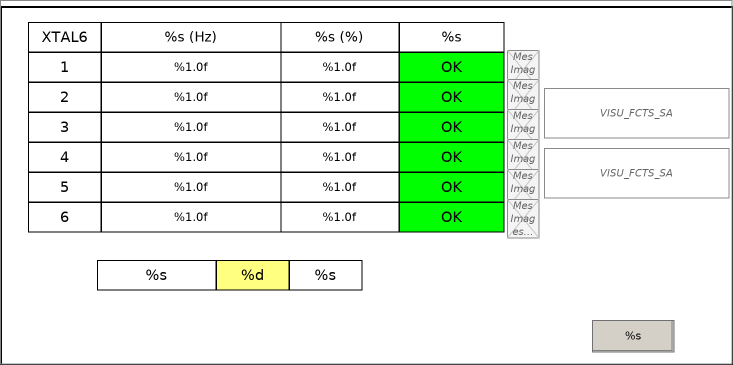
VISUALIZATION VISU_XTAL6_ZOOM  // 733x365, background image fond_blanc_1280_1024
VAR_IN_OUT
	m_Input_XTAL6 : BLOCK_XTAL6;
END_VAR
    Rectangle (0,6 733x359)
    RoundedRectangle (280,52 119x30), "%1.0f", text variable: m_Input_XTAL6.STATE_LIFE[1]
    RoundedRectangle (280,82 119x30), "%1.0f", text variable: m_Input_XTAL6.STATE_LIFE[2]
    RoundedRectangle (280,112 119x30), "%1.0f", text variable: m_Input_XTAL6.STATE_LIFE[3]
    RoundedRectangle (28,52 73x30), "1"
    RoundedRectangle (28,82 73x30), "2"
    RoundedRectangle (28,112 73x30), "3"
    RoundedRectangle (280,22 119x30), "%s (%)", text list: 'TextList_IC6', text index: 13
    RoundedRectangle (399,22 105x30), "%s", text list: 'TextList_IC6', text index: 14
    RoundedRectangle (399,52 105x30), "FAIL", invisible if: NOT m_Input_XTAL6.STATE_QF1
    RoundedRectangle (399,52 105x30), "OK", invisible if: (m_Input_XTAL6.STATE_QF1) <> 0
    RoundedRectangle (399,82 105x30), "FAIL", invisible if: NOT m_Input_XTAL6.STATE_QF2
    RoundedRectangle (399,82 105x30), "OK", invisible if: (m_Input_XTAL6.STATE_QF2) <> 0
    RoundedRectangle (399,112 105x30), "FAIL", invisible if: NOT m_Input_XTAL6.STATE_QF3
    RoundedRectangle (399,112 105x30), "OK", invisible if: (m_Input_XTAL6.STATE_QF3) <> 0
    RoundedRectangle (280,142 119x30), "%1.0f", text variable: m_Input_XTAL6.STATE_LIFE[4]
    RoundedRectangle (280,172 119x30), "%1.0f", text variable: m_Input_XTAL6.STATE_LIFE[5]
    RoundedRectangle (280,202 119x30), "%1.0f", text variable: m_Input_XTAL6.STATE_LIFE[6]
    RoundedRectangle (28,142 73x30), "4"
    RoundedRectangle (28,172 73x30), "5"
    RoundedRectangle (28,202 73x30), "6"
    RoundedRectangle (399,142 105x30), "FAIL", invisible if: NOT m_Input_XTAL6.STATE_QF4
    RoundedRectangle (399,142 105x30), "OK", invisible if: (m_Input_XTAL6.STATE_QF4) <> 0
    RoundedRectangle (399,172 105x30), "FAIL", invisible if: NOT m_Input_XTAL6.STATE_QF5
    RoundedRectangle (399,172 105x30), "OK", invisible if: (m_Input_XTAL6.STATE_QF5) <> 0
    RoundedRectangle (399,202 105x30), "FAIL", invisible if: NOT m_Input_XTAL6.STATE_QF6
    RoundedRectangle (399,202 105x30), "OK", invisible if: (m_Input_XTAL6.STATE_QF6) <> 0
    RoundedRectangle (28,22 73x30), "XTAL6"
    RoundedRectangle (97,260 119x30), "%s", text list: 'TextList_SA_Operations', text index: 23
    RoundedRectangle (216,260 73x30), "%d", text variable: m_Input_XTAL6.PRM_CONS_POSITION_QZ, input disabled if: NOT Global_Variables.PRG_USER.ACTU_USER.MAINTENANCE OR MACHINE.STATE_Prod
        OnMouseDown: write the text variable via VisuDialogs.Numpad, min 1, max 6
    RoundedRectangle (289,260 73x30), "%s", text variable: m_Input_XTAL6.STATE_POSITION
    RoundedRectangle (101,52 180x30), "%1.0f", text variable: m_Input_XTAL6.STATE_FREQUENCY[1]
    RoundedRectangle (101,82 180x30), "%1.0f", text variable: m_Input_XTAL6.STATE_FREQUENCY[2]
    RoundedRectangle (101,112 180x30), "%1.0f", text variable: m_Input_XTAL6.STATE_FREQUENCY[3]
    RoundedRectangle (101,22 180x30), "%s (Hz)", text list: 'TextList_IC6', text index: 12
    RoundedRectangle (101,142 180x30), "%1.0f", text variable: m_Input_XTAL6.STATE_FREQUENCY[4]
    RoundedRectangle (101,172 180x30), "%1.0f", text variable: m_Input_XTAL6.STATE_FREQUENCY[5]
    RoundedRectangle (101,202 180x30), "%1.0f", text variable: m_Input_XTAL6.STATE_FREQUENCY[6]
    Image (507,50 32x39), invisible if: NOT m_Input_XTAL6.ALM_SURV_ACTIVITY_QZ1.DEF AND NOT m_Input_XTAL6.ALM_SURV_LIFE_QZ1.DEF, image: MesImages.warning
    Image (507,79 32x39), invisible if: NOT m_Input_XTAL6.ALM_SURV_ACTIVITY_QZ2.DEF AND NOT m_Input_XTAL6.ALM_SURV_LIFE_QZ2.DEF, image: MesImages.warning
    Image (507,109 32x39), invisible if: NOT m_Input_XTAL6.ALM_SURV_ACTIVITY_QZ3.DEF AND NOT m_Input_XTAL6.ALM_SURV_LIFE_QZ3.DEF, image: MesImages.warning
    Image (507,139 32x39), invisible if: NOT m_Input_XTAL6.ALM_SURV_ACTIVITY_QZ4.DEF AND NOT m_Input_XTAL6.ALM_SURV_LIFE_QZ4.DEF, image: MesImages.warning
    Image (507,169 32x39), invisible if: NOT m_Input_XTAL6.ALM_SURV_ACTIVITY_QZ5.DEF AND NOT m_Input_XTAL6.ALM_SURV_LIFE_QZ5.DEF, image: MesImages.warning
    Image (507,199 32x39), invisible if: NOT m_Input_XTAL6.ALM_SURV_ACTIVITY_QZ6.DEF AND NOT m_Input_XTAL6.ALM_SURV_LIFE_QZ6.DEF, image: MesImages.warning
    Frame (544,88 185x50)
        shows VISU_FCTS_SA(m_Input_ID_XML := 21, m_Input_Operation := m_Input_XTAL6.OP_Scan_Quartz, m_Input_UserRight := PRG_USER.ACTU_USER.FONCTION_SA AND NOT MACHINE.STATE_PROD)
    Frame (544,148 185x50)
        shows VISU_FCTS_SA(m_Input_ID_XML := 22, m_Input_Operation := m_Input_XTAL6.OP_Positionnement, m_Input_UserRight := PRG_USER.ACTU_USER.FONCTION_SA AND NOT MACHINE.STATE_PROD)
    Button (592,320 82x32), "%s", text list: 'TextList_Basiques', text index: 8
        OnMouseClick: change screen: Previous 
        OnMouseClick: execute { .VISU_INDEX_MANU := 0; }
END_VISUALIZATION

(* stored: Version 1.1.0.1, ProductVersion 3.1.4024.10
   Visu VISU_XTAL6_ZOOM: Id {bb015895-8243-408c-b06a-f705a07ed475} *)
